DATA_BLOCK "Global_Vars"
{ S7_Optimized_Access := 'TRUE' }
VERSION : 0.1
   VAR
      Progr : Array[0..999] of "typeProgrDefinition"; // Renamed from Articles
   END_VAR
BEGIN

END_DATA_BLOCK
